// TIA Portal V17 export
// export: Created 2026-04-13T11:12:41.6412663Z, ExportSetting WithDefaults, DisplayName Totally Integrated Automation Portal, DisplayVersion V17 Update 4, DisplayName TIA Portal Openness, DisplayVersion V17 Update 4, DisplayName TIA Portal Version Control Interface, DisplayVersion V17, DisplayName SINAMICS Startdrive Advanced, DisplayVersion V17, DisplayName SINAMICS Startdrive G130, G150, S120, S150, SINAMICS MV, S210, DisplayVersion V17, DisplayName SINAMICS Startdrive G110M, G120, G120C, G120D, G120P, G115D, DisplayVersion V17, DisplayName STEP 7 Professional, DisplayVersion V17 Update 4, DisplayName STEP 7 Safety, DisplayVersion V17, DisplayName WinCC Professional, DisplayVersion V17 Update 4
FUNCTION_BLOCK "A8-阀开关报警"   // FB37, SCL
{ S7_Optimized_Access := 'TRUE' }
VERSION : 0.1
// stored: AutoNumber true, IsIECCheckEnabled false, IsRetainMemResEnabled false, MemoryReserve 100, SetENOAutomatically false, UDAEnableTagReadback false
   VAR_OUTPUT
      阀开报警 : Bool;
      阀关报警 : Bool;
   END_VAR
   VAR_IN_OUT
      阀状态 : Bool;
      阀开信号 : Bool;
      阀关信号 : Bool;
   END_VAR
   VAR
      TON1 : TON_TIME;
      TON2 { S7_SetPoint := 'True'} : TON_TIME;
   END_VAR
BEGIN
   #TON1(IN := #"阀状态" AND NOT #"阀开信号",
         PT := T#10s,
         Q => #"阀开报警");
   IF NOT #"阀状态" THEN

       #"阀开报警" := FALSE;
   END_IF;


   #TON2(IN := #"阀状态" = FALSE AND NOT #"阀关信号",
         PT := T#10s,
         Q => #"阀关报警");
   IF #"阀状态" THEN

       #"阀关报警" := FALSE;
   END_IF;
END_FUNCTION_BLOCK
